Fanuc KAREL source: NC0007.KL

PROGRAM NC0007
%NOLOCKGROUP
ROUTINE R
VAR
S1:INTEGER
BEGIN
S1=1
IF (S1=1) THEN
IF (S1=1) THEN
IF (S1=1) THEN
IF (S1=1) THEN
IF (S1=1) THEN
IF (S1=1) THEN
IF (S1=1) THEN
IF (S1=1) THEN
IF (S1=1) THEN
IF (S1=1) THEN
S1=(S1+1)
ELSE
S1=(S1+2)
ENDIF
ELSE
S1=(S1+2)
ENDIF
ELSE
S1=(S1+2)
ENDIF
ELSE
S1=(S1+2)
ENDIF
ELSE
S1=(S1+2)
ENDIF
ELSE
S1=(S1+2)
ENDIF
ELSE
S1=(S1+2)
ENDIF
ELSE
S1=(S1+2)
ENDIF
ELSE
S1=(S1+2)
ENDIF
ELSE
S1=(S1+2)
ENDIF
END R
BEGIN
R
END NC0007
